(* PLC project SafeLOGIC-1, BrAutomation SafeDESIGNER  4.3.4.4 *)
(* stored: companyURL http://www.br-automation.com, creationDateTime Thu Jun 24 15:45:45 2021 *)

PROGRAM Main
  VAR  (* added by the conversion: wires and edge detectors of the diagram *)
    _SAFEBOOL_TO_BOOL50_OUT : BOOL;
  END_VAR

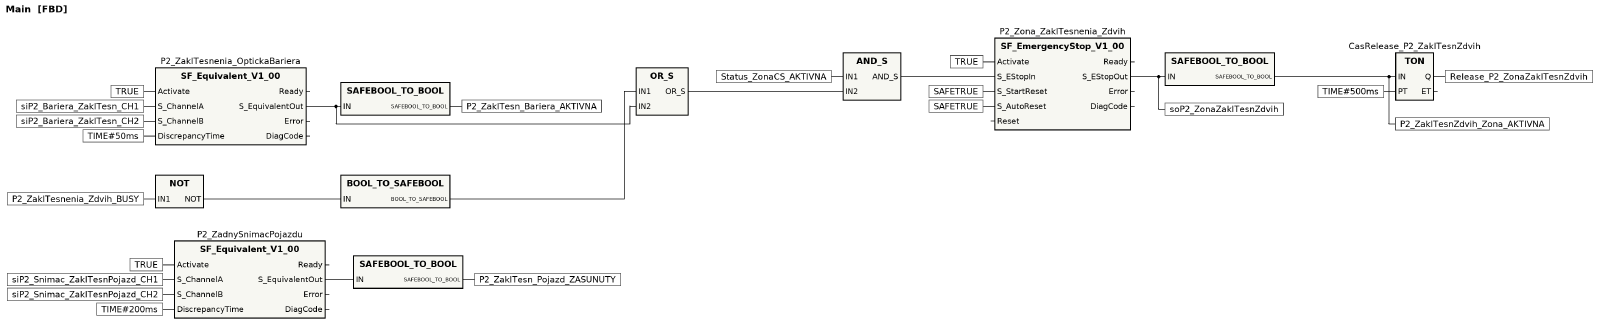
(* FBD diagram, written out as Structured Text *)
P2_ZaklTesnenia_OptickaBariera(Activate := TRUE, S_ChannelA := siP2_Bariera_ZaklTesn_CH1, S_ChannelB := siP2_Bariera_ZaklTesn_CH2, DiscrepancyTime := TIME#50ms);
P2_Zona_ZaklTesnenia_Zdvih(Activate := TRUE, S_EStopIn := AND_S(Status_ZonaCS_AKTIVNA, OR_S(BOOL_TO_SAFEBOOL(NOT P2_ZaklTesnenia_Zdvih_BUSY), P2_ZaklTesnenia_OptickaBariera.S_EquivalentOut)), S_StartReset := SAFETRUE, S_AutoReset := SAFETRUE);
soP2_ZonaZaklTesnZdvih := P2_Zona_ZaklTesnenia_Zdvih.S_EStopOut;
_SAFEBOOL_TO_BOOL50_OUT := SAFEBOOL_TO_BOOL(P2_Zona_ZaklTesnenia_Zdvih.S_EStopOut);
P2_ZaklTesnZdvih_Zona_AKTIVNA := _SAFEBOOL_TO_BOOL50_OUT;
CasRelease_P2_ZaklTesnZdvih(IN := _SAFEBOOL_TO_BOOL50_OUT, PT := TIME#500ms);
Release_P2_ZonaZaklTesnZdvih := CasRelease_P2_ZaklTesnZdvih.Q;
P2_ZaklTesn_Bariera_AKTIVNA := SAFEBOOL_TO_BOOL(P2_ZaklTesnenia_OptickaBariera.S_EquivalentOut);
P2_ZadnySnimacPojazdu(Activate := TRUE, S_ChannelA := siP2_Snimac_ZaklTesnPojazd_CH1, S_ChannelB := siP2_Snimac_ZaklTesnPojazd_CH2, DiscrepancyTime := TIME#200ms);
P2_ZaklTesn_Pojazd_ZASUNUTY := SAFEBOOL_TO_BOOL(P2_ZadnySnimacPojazdu.S_EquivalentOut);
END_PROGRAM
